{attribute 'hide_all_locals'}
FUNCTION_BLOCK FB_Car EXTENDS FB_LinkedList_Node IMPLEMENTS ITF_Car

VAR
	Locked:		BOOL;
END_VAR

METHOD FB_init : BOOL
VAR_INPUT
	bInitRetains : 	BOOL; // if TRUE, the retain variables are initialized (warm start / cold start)
	bInCopyCode : 	BOOL;  // if TRUE, the instance afterwards gets moved into the copy code (online change)
END_VAR
p_LinkMaster := MAIN.fbCarFleet;
END_METHOD

{attribute 'monitoring' := 'call'}
PROPERTY p_Locked : BOOL
GET
p_Locked := Locked;
END_GET
SET
Locked := p_Locked;
END_SET
END_PROPERTY

END_FUNCTION_BLOCK

(* stored: Version 1.1.0.1, ProductVersion 3.1.4024.12
   POU FB_Car: Id {f48c1ede-733f-42f9-90bd-fec45d9a843c}, SpecialFunc None
   Method FB_init: Id {c1871cd6-aecc-4b40-b7ea-f830c857e06f}
   Property p_Locked: Id {383cc081-e986-4e8b-8019-1ff2809dc156}
   Get Get: Id {f416bf3c-1616-48df-85b4-84cdf418be81}
   Set Set: Id {0a2a5928-5d97-4a74-865b-dae9e6f089e9} *)
